FUNCTION_BLOCK FB_Busy2
VAR_INPUT
	bSens	 :BOOL;
	tBusy	 :TIME;
	tFree	 :TIME;
	Reset	 :BOOL;
END_VAR
VAR_OUTPUT
	ConvBusy :BOOL;
END_VAR
VAR
	Timer1	 :TON;
	Timer2	 :TON;
END_VAR

Timer1 (IN := 	  bSens, PT := tBusy);
IF Timer1.Q THEN ConvBusy := TRUE;
END_IF
Timer2 (IN := NOT bSens, PT := tFree);
IF Timer2.Q (*OR Reset*) THEN ConvBusy := FALSE;
END_IF

END_FUNCTION_BLOCK

(* stored: Version 1.1.0.1, ProductVersion 3.1.4024.4
   POU FB_Busy2: Id {192239bf-b071-4671-970b-cb6c0c703943}, SpecialFunc None *)
